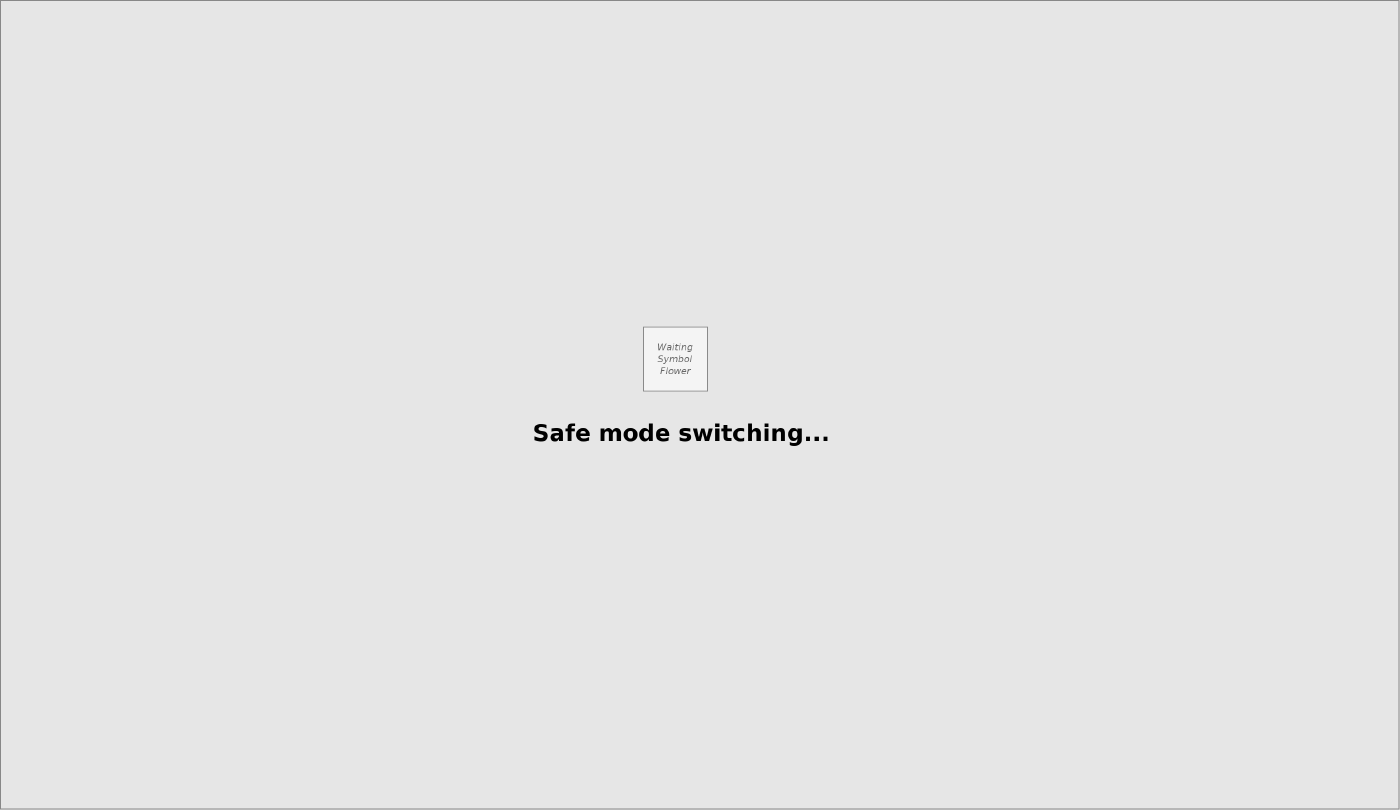
VISUALIZATION PageSwitchMode_1  // 1520x880
    Label (490,450 500x40), "Safe mode switching..."
    WaitingSymbolFlower (698,355 70x70)
END_VISUALIZATION

(* stored: Version 1.1.0.1, ProductVersion 3.1.4024.12
   Visu PageSwitchMode_1: Id {a30ef58a-28c2-4b98-8917-5da9cc4081ff} *)
